FUNCTION_BLOCK GPIOChip (* Service Interface Function Block Type *)
  (* Description: Copyright (c) 2023 OFFIS e.V. This program and the accompanying materials are made available under the terms of the Eclipse Public License 2.0 which is available at https://www.eclipse.org/legal/epl-2.0/ SPDX-License-Identifier: EPL-2.0 *)
  (* Version 3.0, 2025-04-14, Patrick Aigner, changed package *)
  (* Version 1.0, 2023-11-10, Jörg Walter, OFFIS e.V. *)
  PACKAGE eclipse4diac::io::gpiochip;
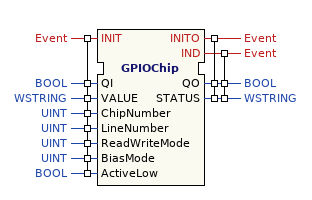
  EVENT_INPUT
    INIT WITH QI, VALUE, ChipNumber, LineNumber, ReadWriteMode, BiasMode, ActiveLow; (* Service Initialization *)
  END_EVENT
  EVENT_OUTPUT
    INITO WITH QO, STATUS; (* Initialization Confirm *)
    IND WITH QO, STATUS; (* Indication from Resource *)
  END_EVENT
  VAR_INPUT
    QI : BOOL; (* Event Input Qualifier *)
    VALUE : WSTRING; (* Receiver IX/QX block name *)
    ChipNumber : UINT := 0; (* ID of /dev/gpiochipX device *)
    LineNumber : UINT := 0; (* ID of GPIO line within selected chip *)
    ReadWriteMode : UINT := 0; (* Reading/Writing mode of line (0=read, 1=write push/pull, 2=open drain, 3=open source) *)
    BiasMode : UINT := 0; (* Bias mode of line (0=none, 1=pull up, 2=pull down) *)
    ActiveLow : BOOL := 0; (* True if a logic 1 corresponds to low voltage *)
  END_VAR
  VAR_OUTPUT
    QO : BOOL; (* Event Output Qualifier *)
    STATUS : WSTRING; (* Service Status *)
  END_VAR
  SERVICE APPLICATION/RESOURCE
    SEQUENCE normal_establishment
      APPLICATION.INIT+(PARAMS) -> RESOURCE.initialize(PARAMS) -> APPLICATION.INITO+();
    END_SEQUENCE
    SEQUENCE unsuccessful_establishment
      APPLICATION.INIT+(PARAMS) -> RESOURCE.initialize(PARAMS) -> APPLICATION.INITO-(STATUS);
    END_SEQUENCE
  END_SERVICE
END_FUNCTION_BLOCK
